Universal Robots URScript: 00C_06_BoXian_ToZero.script

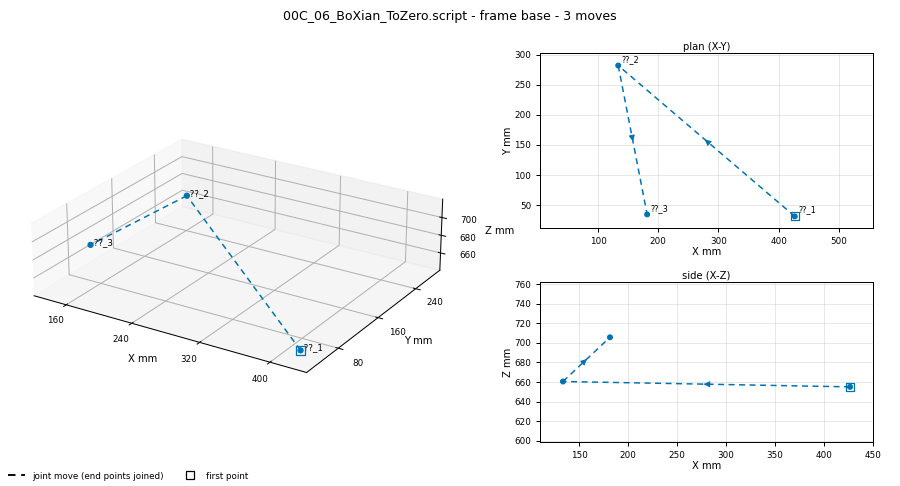
[picture p0: tool path of 00C_06_BoXian_ToZero.script in frame base, 3 of 3 moves have a stored position in this frame; points joined in program order, loops and branches not executed]
def P00C_06_BoXian_ToZero():
  set_standard_analog_input_domain(0, 1)
  set_standard_analog_input_domain(1, 1)
  set_tool_analog_input_domain(0, 1)
  set_tool_analog_input_domain(1, 1)
  set_analog_outputdomain(0, 0)
  set_analog_outputdomain(1, 0)
  set_tool_voltage(0)
  set_input_actions_to_default()
  set_tcp(p[-0.06448999999999999,0.0207,0.28314999999999996,0.0,0.0,1.5902])
  set_payload(8.0)
  set_safety_mode_transition_hardness(1)
  set_gravity([0.0, 0.0, 9.82])
  $ 1 "机器人程序"
  $ 2 "MoveJ"
  $ 3 "路点_1"
  set_tcp(p[-8.5E-4,0.01448,0.31003,0.0,0.0,-0.3645])
  movej(get_inverse_kin(p[.426773524788, .031349745872, .655059670374, -.007851311721, .061521685542, -1.299004086998], qnear=[0.5012286305427551, -1.4666112104998987, -2.670898977910177, -0.6036627928363245, -1.5242565313922327, -3.0075951258288782]), a=0.6981317007977318, v=0.5235987755982988)
  $ 4 "路点_2"
  set_tcp(p[-8.5E-4,0.01448,0.31003,0.0,0.0,-0.3645])
  movej(get_inverse_kin(p[.133482221842, .281881306661, .660550846213, -.046045832543, .049046162551, .006739020603], qnear=[1.7449462413787842, -1.0578840414630335, -2.853910032902853, -0.836402718220846, -1.515174690877096, -2.944904390965597]), a=0.6981317007977318, v=0.5235987755982988)
  $ 5 "路点_3"
  set_tcp(p[-8.5E-4,0.01448,0.31003,0.0,0.0,-0.3645])
  movej(get_inverse_kin(p[.181508728915, .034600708981, .705736457852, .017025264227, .054065104184, -1.587634587539], qnear=[1.6280419826507568, 0.05510425567626953, -2.8315115610705774, -1.8881552855121058, -1.548361603413717, -4.4239166418658655]), a=0.6981317007977318, v=0.5235987755982988)
end
